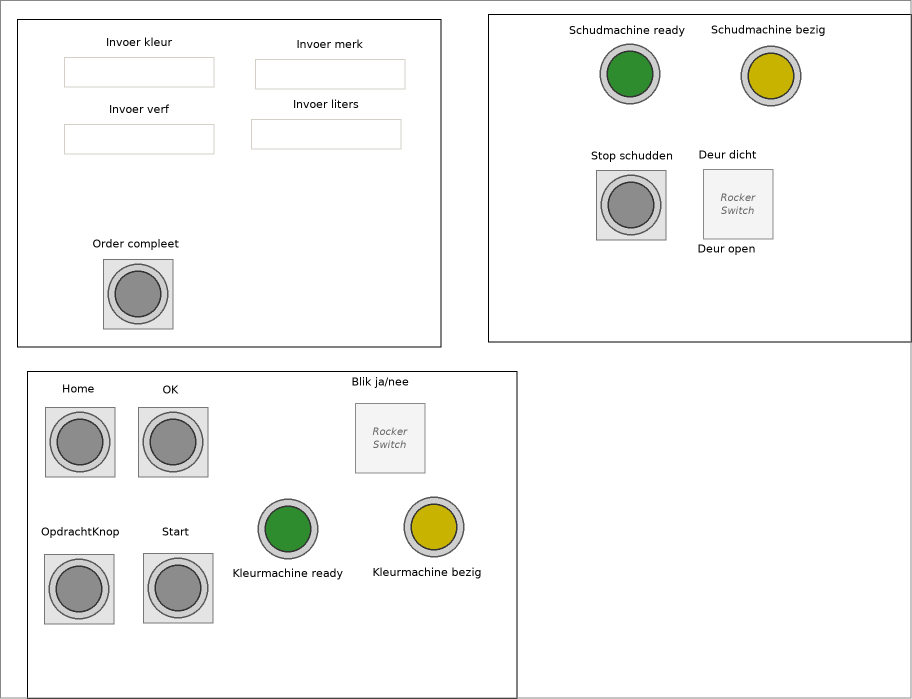
VISUALIZATION Visu_main  // 912x699
    Rectangle (488,14 424x328)
    Rectangle (17,19 424x328)
    Textfield (64,57 150x30)
        OnMouseClick: write GVL.kleurVerf via Edit
    Lamp1 (595,39 70x70), variable: schudmachine.schudmachineReady, style: Lamp-Lamp1-Green
    PushSwitch (596,170 70x70), variable: schudmachine.stopSchudden, behaviour: TAP, style: Switch-PushSwitch-Gray
    RockerSwitch (703,169 70x70), variable: schudmachine.deurDicht, behaviour: TOGGLE, style: Switch-RockerSwitch-Gray
    Label (677,140 101x30), "Deur dicht"
    Label (579,141 106x30), "Stop schudden"
    Label (676,234 101x30), "Deur open"
    Lamp1 (736,41 70x70), variable: schudmachine.schudMachineBezig, style: Lamp-Lamp1-Yellow
    Label (563,13 128x35), "Schudmachine ready"
    Label (702,15 133x30), "Schudmachine bezig"
    Label (75,25 128x35), "Invoer kleur"
    Textfield (255,59 150x30)
        OnMouseClick: write GVL.merkVerf via Edit
    Label (266,27 128x35), "Invoer merk"
    Textfield (64,124 150x30)
        OnMouseClick: write GVL.typeVerf via Edit
    Label (75,92 128x35), "Invoer verf"
    Textfield (251,119 150x30)
        OnMouseClick: write GVL.hoeveelVerf via Edit
    Label (262,87 128x35), "Invoer liters"
    PushSwitch (103,259 70x70), variable: Medewerker.orderCompleet, behaviour: TAP, style: Switch-PushSwitch-Gray
    Label (83,229 106x30), "Order compleet"
    Rectangle (27,371 490x328)
    PushSwitch (45,407 70x70), variable: GVL.homeKnop, behaviour: TAP, style: Switch-PushSwitch-Gray
    PushSwitch (138,407 70x70), variable: GVL.okeKnop, behaviour: TAP, style: Switch-PushSwitch-Gray
    RockerSwitch (355,403 70x70), variable: GVL.blikPresent, behaviour: TOGGLE, style: Switch-RockerSwitch-Gray
    Label (39,374 79x30), "Home"
    Label (131,375 79x30), "OK"
    Label (341,367 79x30), "Blik ja/nee"
    PushSwitch (44,554 70x70), variable: GVL.opdrachtKnop, behaviour: TAP, style: Switch-PushSwitch-Gray
    PushSwitch (143,553 70x70), variable: GVL.startKnop, behaviour: TAP, style: Switch-PushSwitch-Gray
    Label (41,517 79x30), "OpdrachtKnop"
    Label (136,517 79x30), "Start"
    Lamp1 (253,494 70x70), variable: kleurmachine.kleurmachineReady, style: Lamp-Lamp1-Green
    Lamp1 (399,492 70x70), variable: kleurmachine.kleurmachineBezig, style: Lamp-Lamp1-Yellow
    Label (224,556 128x35), "Kleurmachine ready"
    Label (363,555 128x35), "Kleurmachine bezig"
END_VISUALIZATION

(* stored: Version 1.1.0.1, ProductVersion 3.1.4024.15
   Visu Visu_main: Id {8a145de3-b456-450d-9a14-c034f53585d6} *)
